FUNCTION_BLOCK XtsHardware
VAR
END_VAR

METHOD CheckModuleVoltages : BOOL
VAR_INPUT
END_VAR
END_METHOD

METHOD GetTrackLength : BOOL
VAR_INPUT
END_VAR
END_METHOD

END_FUNCTION_BLOCK

(* stored: Version 1.1.0.1, ProductVersion 3.1.4024.12
   POU XtsHardware: Id {bacf700d-de35-4e0b-aeba-07a502dd8b3e}, SpecialFunc None
   Method CheckModuleVoltages: Id {4672f55d-f08e-44da-ac15-11867e254a29}
   Method GetTrackLength: Id {c743714e-2a5a-4dcf-b1d5-677b958f5b53} *)
